TYPE ST_Chamber1SpinAxisMoveAbsParam :
STRUCT
	Position : LREAL;
	Velocity : LREAL;
	Acceleration : LREAL;
	Deceleration : LREAL;
END_STRUCT
END_TYPE

(* stored: Version 1.1.0.1, ProductVersion 3.1.4026.18
   DUT ST_Chamber1SpinAxisMoveAbsParam: Id {9e809cb0-9869-41cb-83b7-96945d386765} *)
